% RSLogix 500 project INTRO TO PLC - JOB 22.RSS, saved by version 10.00.00.00 %
PROJECT "PL06B"    % processor: Bul.1763 MicroLogix 1100 Series B %

PROGRAM FILES
  LAD 2   21 rungs

DATA FILES
  O0 OUTPUT  4 elements
  I1 INPUT  6 elements
  S2 STATUS  66 elements
  B3 BINARY  1 elements
  T4 TIMER  10 elements
  C5 COUNTER  3 elements
  R6 CONTROL  1 elements
  N7 INTEGER  5 elements
  F8 FLOAT  1 elements

LADDER 2
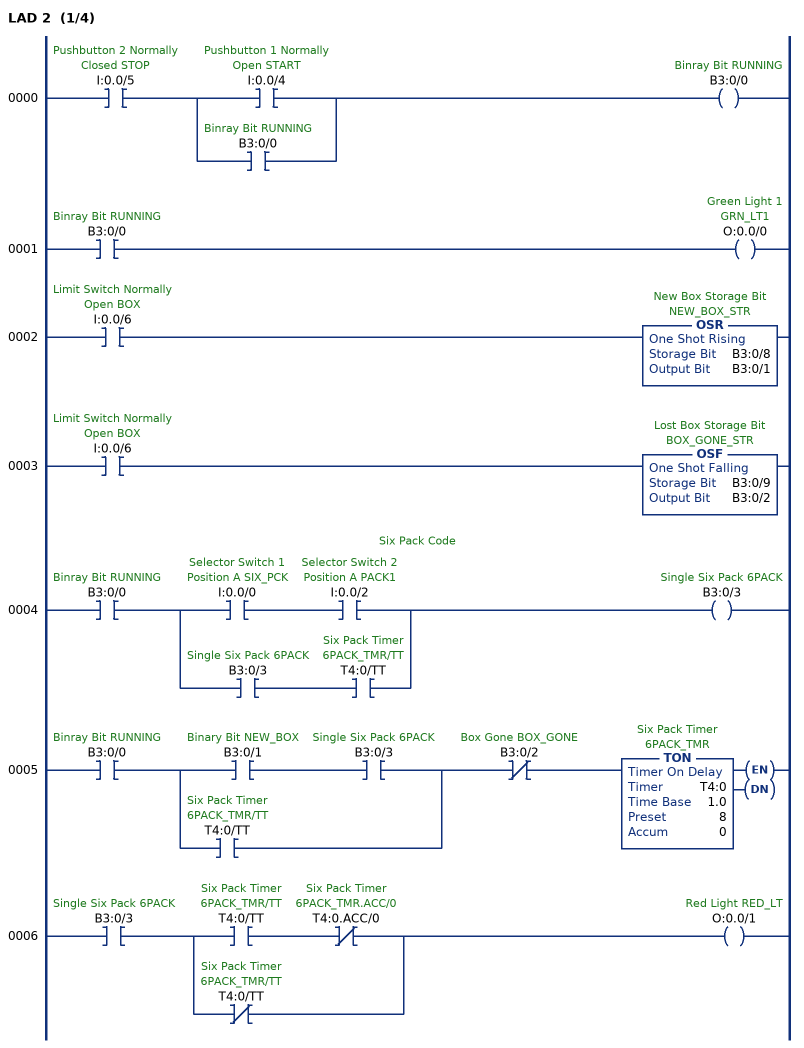
% Rung: 0 %
SOR XIC I:0.0/5 BST XIC I:0.0/4 NXB XIC B3:0/0 BND OTE B3:0/0 EOR
%   I:0.0/5  STOP  "Pushbutton 2 Normally Closed" %
%   I:0.0/4  START  "Pushbutton 1 Normally Open" %
%   B3:0/0  RUNNING  "Binray Bit" %
% Rung: 1 %
SOR XIC B3:0/0 OTE O:0.0/0 EOR
%   B3:0/0  RUNNING  "Binray Bit" %
%   O:0.0/0  GRN_LT1  "Green Light 1" %
% Rung: 2 %
SOR XIC I:0.0/6 OSR B3:0/8 B3:0/1 EOR
%   I:0.0/6  BOX  "Limit Switch Normally Open" %
%   B3:0/8  NEW_BOX_STR  "New Box Storage Bit" %
%   B3:0/1  NEW_BOX  "Binary Bit" %
% Rung: 3 %
SOR XIC I:0.0/6 OSF B3:0/9 B3:0/2 EOR
%   I:0.0/6  BOX  "Limit Switch Normally Open" %
%   B3:0/9  BOX_GONE_STR  "Lost Box Storage Bit" %
%   B3:0/2  BOX_GONE  "Box Gone" %
% Rung: 4 %
% Six Pack Code %
SOR XIC B3:0/0 BST XIC I:0.0/0 XIC I:0.0/2 NXB XIC B3:0/3 XIC T4:0/TT BND OTE B3:0/3 EOR
%   B3:0/0  RUNNING  "Binray Bit" %
%   I:0.0/0  SIX_PCK  "Selector Switch 1 Position A" %
%   I:0.0/2  PACK1  "Selector Switch 2 Position A" %
%   B3:0/3  6PACK  "Single Six Pack" %
%   T4:0  6PACK_TMR  "Six Pack Timer" %
% Rung: 5 %
SOR XIC B3:0/0 BST XIC B3:0/1 XIC B3:0/3 NXB XIC T4:0/TT BND XIO B3:0/2 TON T4:0 1.0 8 0 EOR
%   B3:0/0  RUNNING  "Binray Bit" %
%   B3:0/1  NEW_BOX  "Binary Bit" %
%   B3:0/3  6PACK  "Single Six Pack" %
%   T4:0  6PACK_TMR  "Six Pack Timer" %
%   B3:0/2  BOX_GONE  "Box Gone" %
% Rung: 6 %
SOR XIC B3:0/3 BST XIC T4:0/TT XIO T4:0.ACC/0 NXB XIO T4:0/TT BND OTE O:0.0/1 EOR
%   B3:0/3  6PACK  "Single Six Pack" %
%   T4:0  6PACK_TMR  "Six Pack Timer" %
%   O:0.0/1  RED_LT  "Red Light" %

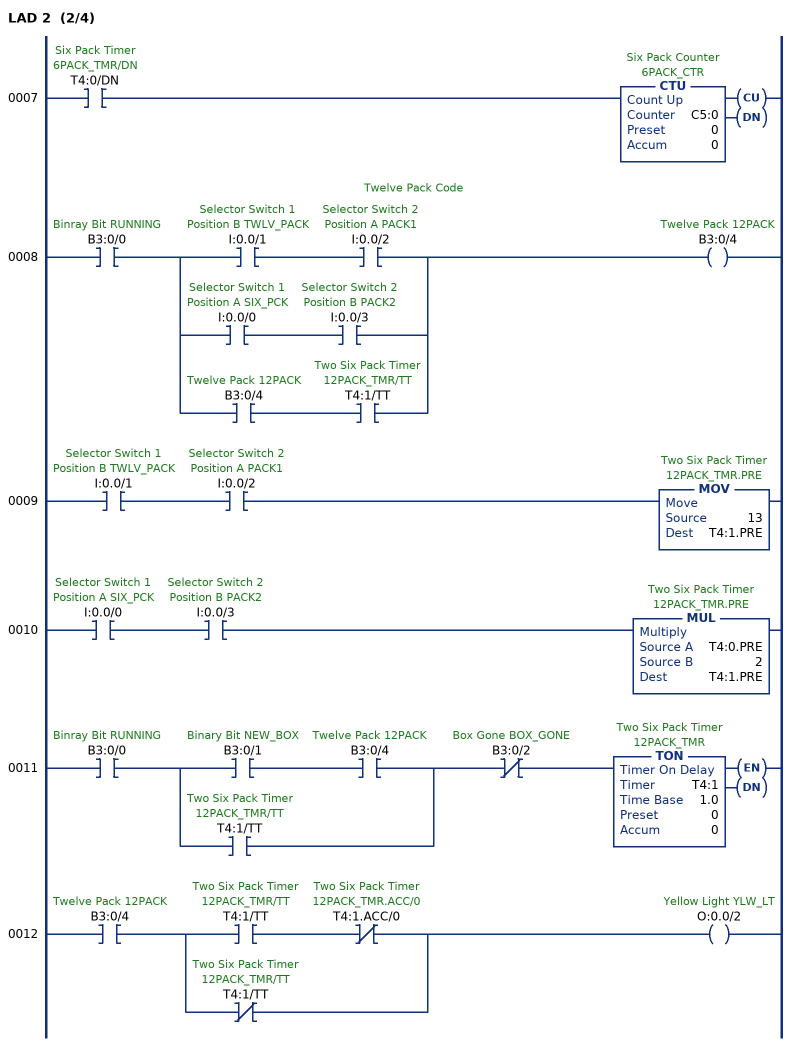
% Rung: 7 %
SOR XIC T4:0/DN CTU C5:0 0 0 EOR
%   T4:0  6PACK_TMR  "Six Pack Timer" %
%   C5:0  6PACK_CTR  "Six Pack Counter" %
% Rung: 8 %
% Twelve Pack Code %
SOR XIC B3:0/0 BST XIC I:0.0/1 XIC I:0.0/2 NXB XIC I:0.0/0 XIC I:0.0/3 NXB XIC B3:0/4 XIC T4:1/TT BND OTE B3:0/4 EOR
%   B3:0/0  RUNNING  "Binray Bit" %
%   I:0.0/1  TWLV_PACK  "Selector Switch 1 Position B" %
%   I:0.0/2  PACK1  "Selector Switch 2 Position A" %
%   I:0.0/0  SIX_PCK  "Selector Switch 1 Position A" %
%   I:0.0/3  PACK2  "Selector Switch 2 Position B" %
%   B3:0/4  12PACK  "Twelve Pack" %
%   T4:1  12PACK_TMR  "Two Six Pack Timer" %
% Rung: 9 %
SOR XIC I:0.0/1 XIC I:0.0/2 MOV 13 T4:1.PRE EOR
%   I:0.0/1  TWLV_PACK  "Selector Switch 1 Position B" %
%   I:0.0/2  PACK1  "Selector Switch 2 Position A" %
%   T4:1  12PACK_TMR  "Two Six Pack Timer" %
% Rung: 10 %
SOR XIC I:0.0/0 XIC I:0.0/3 MUL T4:0.PRE 2 T4:1.PRE EOR
%   I:0.0/0  SIX_PCK  "Selector Switch 1 Position A" %
%   I:0.0/3  PACK2  "Selector Switch 2 Position B" %
%   T4:0  6PACK_TMR  "Six Pack Timer" %
%   T4:1  12PACK_TMR  "Two Six Pack Timer" %
% Rung: 11 %
SOR XIC B3:0/0 BST XIC B3:0/1 XIC B3:0/4 NXB XIC T4:1/TT BND XIO B3:0/2 TON T4:1 1.0 0 0 EOR
%   B3:0/0  RUNNING  "Binray Bit" %
%   B3:0/1  NEW_BOX  "Binary Bit" %
%   B3:0/4  12PACK  "Twelve Pack" %
%   T4:1  12PACK_TMR  "Two Six Pack Timer" %
%   B3:0/2  BOX_GONE  "Box Gone" %
% Rung: 12 %
SOR XIC B3:0/4 BST XIC T4:1/TT XIO T4:1.ACC/0 NXB XIO T4:1/TT BND OTE O:0.0/2 EOR
%   B3:0/4  12PACK  "Twelve Pack" %
%   T4:1  12PACK_TMR  "Two Six Pack Timer" %
%   O:0.0/2  YLW_LT  "Yellow Light" %

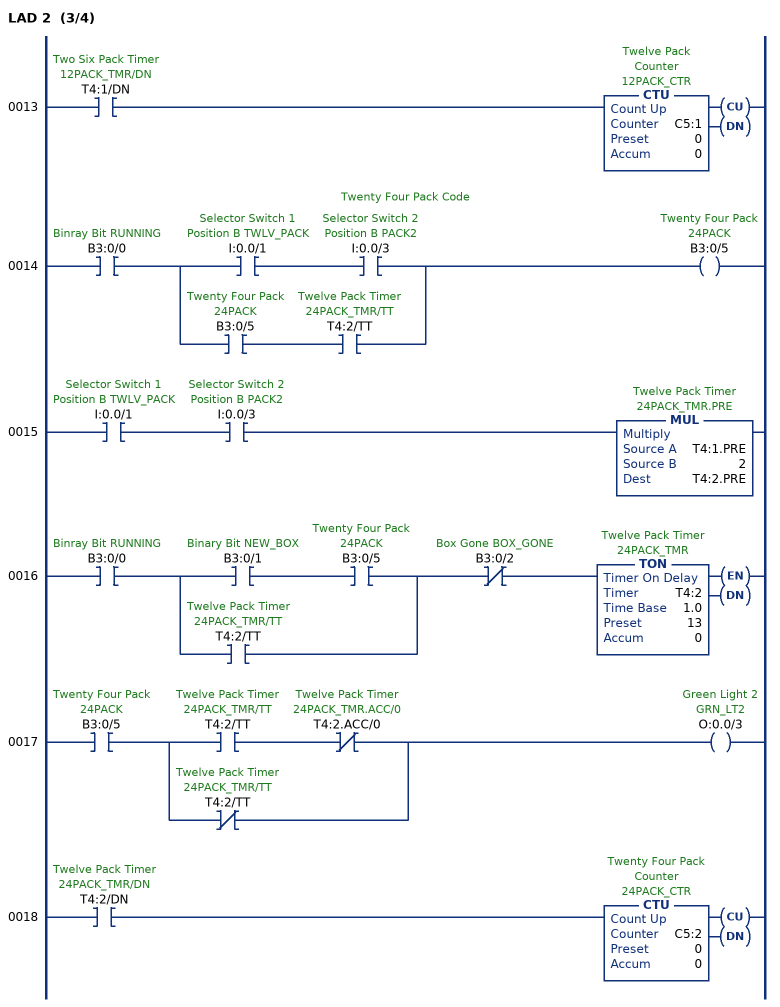
% Rung: 13 %
SOR XIC T4:1/DN CTU C5:1 0 0 EOR
%   T4:1  12PACK_TMR  "Two Six Pack Timer" %
%   C5:1  12PACK_CTR  "Twelve Pack Counter" %
% Rung: 14 %
% Twenty Four Pack Code %
SOR XIC B3:0/0 BST XIC I:0.0/1 XIC I:0.0/3 NXB XIC B3:0/5 XIC T4:2/TT BND OTE B3:0/5 EOR
%   B3:0/0  RUNNING  "Binray Bit" %
%   I:0.0/1  TWLV_PACK  "Selector Switch 1 Position B" %
%   I:0.0/3  PACK2  "Selector Switch 2 Position B" %
%   B3:0/5  24PACK  "Twenty Four Pack" %
%   T4:2  24PACK_TMR  "Twelve Pack Timer" %
% Rung: 15 %
SOR XIC I:0.0/1 XIC I:0.0/3 MUL T4:1.PRE 2 T4:2.PRE EOR
%   I:0.0/1  TWLV_PACK  "Selector Switch 1 Position B" %
%   I:0.0/3  PACK2  "Selector Switch 2 Position B" %
%   T4:1  12PACK_TMR  "Two Six Pack Timer" %
%   T4:2  24PACK_TMR  "Twelve Pack Timer" %
% Rung: 16 %
SOR XIC B3:0/0 BST XIC B3:0/1 XIC B3:0/5 NXB XIC T4:2/TT BND XIO B3:0/2 TON T4:2 1.0 13 0 EOR
%   B3:0/0  RUNNING  "Binray Bit" %
%   B3:0/1  NEW_BOX  "Binary Bit" %
%   B3:0/5  24PACK  "Twenty Four Pack" %
%   T4:2  24PACK_TMR  "Twelve Pack Timer" %
%   B3:0/2  BOX_GONE  "Box Gone" %
% Rung: 17 %
SOR XIC B3:0/5 BST XIC T4:2/TT XIO T4:2.ACC/0 NXB XIO T4:2/TT BND OTE O:0.0/3 EOR
%   B3:0/5  24PACK  "Twenty Four Pack" %
%   T4:2  24PACK_TMR  "Twelve Pack Timer" %
%   O:0.0/3  GRN_LT2  "Green Light 2" %
% Rung: 18 %
SOR XIC T4:2/DN CTU C5:2 0 0 EOR
%   T4:2  24PACK_TMR  "Twelve Pack Timer" %
%   C5:2  24PACK_CTR  "Twenty Four Pack Counter" %

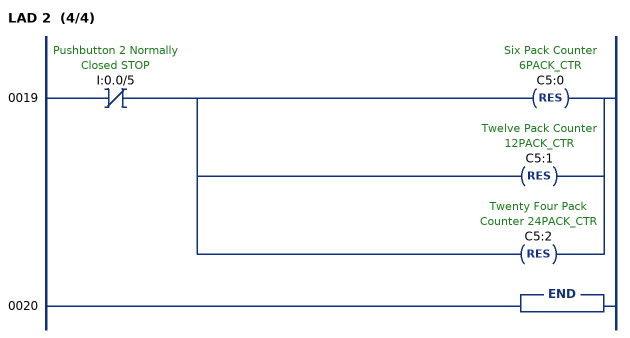
% Rung: 19 %
SOR XIO I:0.0/5 BST RES C5:0 NXB RES C5:1 NXB RES C5:2 BND EOR
%   I:0.0/5  STOP  "Pushbutton 2 Normally Closed" %
%   C5:0  6PACK_CTR  "Six Pack Counter" %
%   C5:1  12PACK_CTR  "Twelve Pack Counter" %
%   C5:2  24PACK_CTR  "Twenty Four Pack Counter" %
% Rung: 20 %
SOR END EOR

OTHER DOCUMENTED ADDRESSES
  B3:0/6  2TWLVPACK  "Two Twelve Packs"
  B3:0/15  SCRATCH  "Scratch Bit"
  B3:1/1  RED_TMR_DNS  "New Box"
  I  
  RTC:0.YR  RTC
  SEL1B  
  T4:3  RST_TMR  "Reset Timer"

DATA TABLE (non-zero values as saved)
DATA B3
% B3:0 % 0X8001
DATA T4
% .PRE .ACC %
% T4:0 % 8 0
% T4:2 % 13 0
% T4:3 % 10 0
DATA N7
% N7:0 % 555 0 0 0 0
